(* CODESYS project INDEX.project

Project tree, tasks and I/O mapping:
  Device : CODESYS Control Win V3, 3S - Smart Software Solutions GmbH, order no. 305021, version 3.5.11.30
    application Application
      libraries: Standard, * (System)
      task MainTask (cyclic, interval t#20ms, priority 1) calls PLC_PRG
      program PLC_PRG [LD]
*)

// Device/Application/PLC_PRG
PROGRAM PLC_PRG
VAR
	TAP1 : BOOL;    // ESTEIRA 1
    TAP2 : BOOL;    // ESTEIRA 2
    S2 : BOOL;      // LIGA
    S0 : BOOL;      // DESLIGA TUDO E RESETA O CONTADOR
    S3 : BOOL;      // SENSOR DE DETECCAO DE PEÇAS
    A : BOOL;       // MOTOR PNEUMATICO
    A1 : BOOL;      // SENSOR MAGNETICO NO FINAL DO CORPO DO CILINDRO
    A0 : BOOL;      // SENSOR MAGNETICO NO COMEÇO DO CORPO DO CILINDRO
	P1: BOOL;
	P2: BOOL;
	P3: BOOL;
	AVANCO : BOOL;
	RETORNO: BOOL;
	P4: BOOL;
	CTU_1: CTU;
	CV1: WORD;
END_VAR

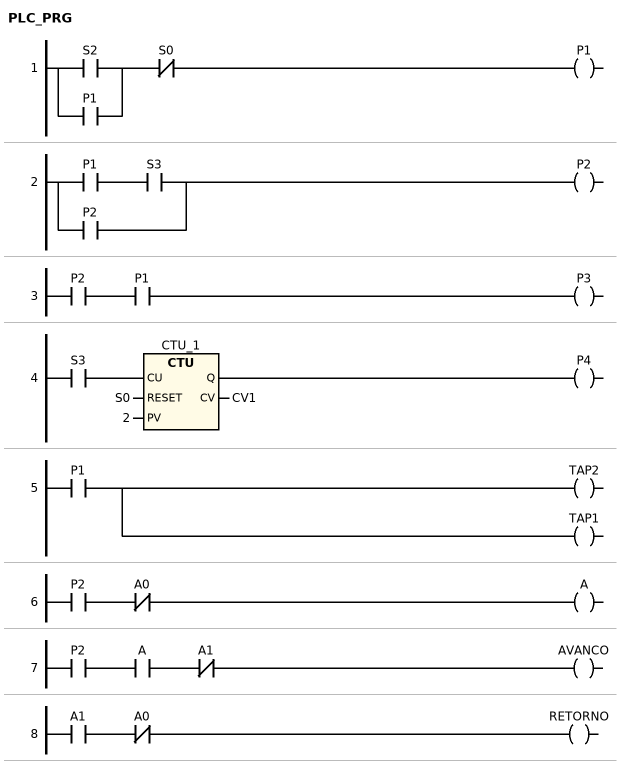
// NETWORK 1
P1 := (S2 OR P1) AND NOT S0;

// NETWORK 2
P2 := P1 AND S3 OR P2;

// NETWORK 3
P3 := P2 AND P1;

// NETWORK 4
CTU_1(CU := S3, RESET := S0, PV := 2, CV => CV1); // CTU
P4 := CTU_1.Q;

// NETWORK 5
TAP2 := P1;
TAP1 := P1;

// NETWORK 6
A := P2 AND NOT A0;

// NETWORK 7
AVANCO := P2 AND A AND NOT A1;

// NETWORK 8
RETORNO := A1 AND NOT A0;

END_PROGRAM
